FUNCTION_BLOCK CHECKPOINT_DISCOVERY (* Composite Function Block Type *)
  (* Standard: 61499-2 *)
  (* Version 0.0, 12/17/2022, Dmitrii, Flexbridge AB, template *)
  PACKAGE UAO.Hackathon;
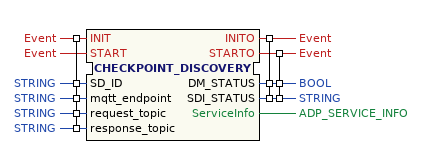
  EVENT_INPUT
    INIT WITH SD_ID, mqtt_endpoint, request_topic, response_topic;
    START;
  END_EVENT
  EVENT_OUTPUT
    INITO WITH SDI_STATUS, DM_STATUS;
    STARTO WITH SDI_STATUS, DM_STATUS;
  END_EVENT
  VAR_INPUT
    SD_ID : STRING;
    mqtt_endpoint : STRING;
    request_topic : STRING;
    response_topic : STRING;
  END_VAR
  VAR_OUTPUT
    DM_STATUS : BOOL;
    SDI_STATUS : STRING; (* Service Status *)
  END_VAR
  PLUGS
    ServiceInfo : ADP_SERVICE_INFO;
  END_PLUGS
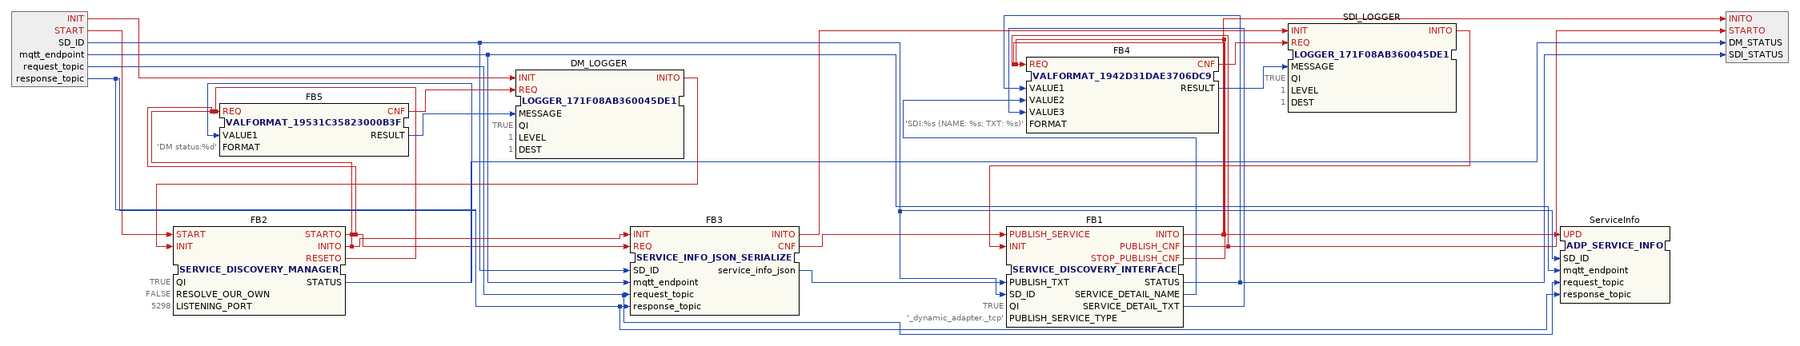
  FBS
    FB1 : SERVICE_DISCOVERY_INTERFACE(QI := TRUE, PUBLISH_SERVICE_TYPE := '_dynamic_adapter._tcp');
    FB2 : SERVICE_DISCOVERY_MANAGER(QI := TRUE, RESOLVE_OUR_OWN := FALSE, LISTENING_PORT := 5298);
    FB3 : SERVICE_INFO_JSON_SERIALIZE;
    DM_LOGGER : LOGGER_171F08AB360045DE1(QI := TRUE, LEVEL := 1, DEST := 1); {SET_ATTRIBUTE(Configuration.GenericFBType.InterfaceParams, Runtime.System#CNT:=1)}
    SDI_LOGGER : LOGGER_171F08AB360045DE1(QI := TRUE, LEVEL := 1, DEST := 1); {SET_ATTRIBUTE(Configuration.GenericFBType.InterfaceParams, Runtime.System#CNT:=1)}
    FB4 : VALFORMAT_1942D31DAE3706DC9(FORMAT := 'SDI:%s (NAME: %s; TXT: %s)'); {SET_ATTRIBUTE(Configuration.GenericFBType.InterfaceParams, Runtime.Standard#I:=3;VALUE${I$}:STRING,STRING,STRING)}
    FB5 : VALFORMAT_19531C35823000B3F(FORMAT := 'DM status:%d'); {SET_ATTRIBUTE(Configuration.GenericFBType.InterfaceParams, Runtime.Standard#I:=1;VALUE${I$}:BOOL)}
  END_FBS
  EVENT_CONNECTIONS
    FB1.INITO TO INITO;
    FB2.STARTO TO FB3.REQ;
    FB3.CNF TO FB1.PUBLISH_SERVICE;
    FB2.INITO TO FB3.INIT;
    START TO FB2.START;
    FB1.INITO TO ServiceInfo.UPD;
    FB1.PUBLISH_CNF TO STARTO;
    INIT TO DM_LOGGER.INIT;
    DM_LOGGER.INITO TO FB2.INIT;
    FB2.INITO TO FB5.REQ;
    FB2.STARTO TO FB5.REQ;
    FB2.RESETO TO FB5.REQ;
    FB3.INITO TO SDI_LOGGER.INIT;
    SDI_LOGGER.INITO TO FB1.INIT;
    FB1.INITO TO FB4.REQ;
    FB1.PUBLISH_CNF TO FB4.REQ;
    FB1.STOP_PUBLISH_CNF TO FB4.REQ;
    FB4.CNF TO SDI_LOGGER.REQ;
    FB5.CNF TO DM_LOGGER.REQ;
  END_CONNECTIONS
  DATA_CONNECTIONS
    mqtt_endpoint TO FB3.mqtt_endpoint;
    request_topic TO FB3.request_topic;
    FB3.service_info_json TO FB1.PUBLISH_TXT;
    SD_ID TO FB3.SD_ID;
    SD_ID TO ServiceInfo.SD_ID;
    SD_ID TO FB1.SD_ID;
    mqtt_endpoint TO ServiceInfo.mqtt_endpoint;
    request_topic TO ServiceInfo.request_topic;
    response_topic TO FB3.response_topic;
    response_topic TO ServiceInfo.response_topic;
    FB2.STATUS TO DM_STATUS;
    FB1.STATUS TO SDI_STATUS;
    FB1.STATUS TO FB4.VALUE1;
    FB1.SERVICE_DETAIL_NAME TO FB4.VALUE2;
    FB1.SERVICE_DETAIL_TXT TO FB4.VALUE3;
    FB4.RESULT TO SDI_LOGGER.MESSAGE;
    FB2.STATUS TO FB5.VALUE1;
    FB5.RESULT TO DM_LOGGER.MESSAGE;
  END_CONNECTIONS
END_FUNCTION_BLOCK
